Yaskawa INFORM job: _DEL197.JBI

/JOB
//NAME _DEL197
//POS
///NPOS 0,0,0,0,0,1
///TOOL 0
///POSTYPE ANGLE
///ANGLE
EX00111=0.0000
//INST
///DATE 2018/11/14 13:43
///ATTR SC,RW,SY
///GROUP1 ST2
///LVARS 5,0,5,0,0,0,0,0
NOP
*top
'live angle st2
GETS PX111 $PX001
GETE LD000 EX111 (1)
DIV LD000 2000
SET LB000 LD000
DOUT OG#(83) LB000
JUMP *top
END
